FUNCTION F_ConfigSubSystemEmulation : BOOL

;

END_FUNCTION

(* stored: Version 1.1.0.1, ProductVersion 3.1.4024.9
   POU F_ConfigSubSystemEmulation: Id {6634f33d-9a62-414a-af75-e09c5fffb480}, SpecialFunc None *)
